Staubli VAL3: TRAJ.pjx

--- TRAJ.pjx ---
Parameters version=s7.5 stackSize=5000 millimeterUnit=true
Program file=changePCircle.pgx
Program file=checkPCircle.pgx
Program file=computeFrame.pgx
Program file=delete.pgx
Program file=deleteItem.pgx
Program file=duplicate.pgx
Program file=find.pgx
Program file=findMove.pgx
Program file=get.pgx
Program file=getDistance.pgx
Program file=getFrame.pgx
Program file=getFrameId.pgx
Program file=getFunctionEdit.pgx
Program file=getFunctionSel.pgx
Program file=getFunctionView.pgx
Program file=getListItem.pgx
Program file=getPoint.pgx
Program file=getSize.pgx
Program file=getSizeItem.pgx
Program file=getTime.pgx
Program file=getTool.pgx
Program file=getTrajItem.pgx
Program file=getTrajType.pgx
Program file=getType.pgx
Program file=goTo.pgx
Program file=HerePoint.pgx
Program file=HerePointCircle.pgx
Program file=insertItem.pgx
Program file=isReachable.pgx
Program file=load.pgx
Program file=loadCycle.pgx
Program file=loadPage.pgx
Program file=makeTraj.pgx
Program file=new.pgx
Program file=onEdit.pgx
Program file=onEditItem.pgx
Program file=onEditTrsf.pgx
Program file=onFunctionEdit.pgx
Program file=onFunctionSel.pgx
Program file=onFunctionView.pgx
Program file=onInsert.pgx
Program file=onProgEnd.pgx
Program file=onRun.pgx
Program file=onSave.pgx
Program file=onStart.pgx
Program file=onStop.pgx
Program file=setFrameId.pgx
Program file=setTool.pgx
Program file=setTrajItem.pgx
Data file=TRAJ.dtx
Library alias=saveData path=Disk://saveData/saveData.pjx
Library alias=page path=Disk://kernel/template/page/page.pjx
Library alias=use path=Disk://kernel/userPage/userPage.pjx
Library alias=language path=Disk://kernel/language/language.pjx
Library alias=tcp path=Disk://kernel/tool/tool.pjx
Library alias=cycleStatus path=Disk://cycleStatus/cycleStatus.pjx
Library alias=pt path=Disk://kernel/template/session/saveTraj/TRAJ/TRAJ.pjx
Type name=TrajectoryItem path=Disk://kernel/template/TrajectoryItem/TrajectoryItem.pjx
Type name=ActionItem path=Disk://kernel/template/ActionItem/ActionItem.pjx
Type name=Trajectory path=Disk://kernel/template/Trajectory/Trajectory.pjx
Type name=InstrItem path=Disk://kernel/template/InstrItem/InstrItem.pjx
Type name=Traies path=Disk://kernel/template/Traies/Traies.pjx
Type name=FrameItem path=Disk://kernel/template/FrameItem/FrameItem.pjx

--- TRAJ.dtx ---
Trajectory tTraj
  [0]
    TrajectoryItem tSuper[3]
      [0]
        num distance
        num moveType = 1
        num nTime
        num nStop
        num nTcpAction
        string comment = "appro"
        bool toStop
        mdesc nom_speed = {tmax=300, rmax=9999, leave=30, reach=30}
        InstrItem iInstr[3]
          [0]
            string sType
            string sData
          [1]
            string sType
            string sData
          [2]
            string sType
            string sData
        num nMoveId
      [1]
        num distance = 2
        num moveType = 1
        num nTime
        num nStop
        num nTcpAction = 2
        string comment = "point"
        bool toStop = true
        mdesc nom_speed = {tmax=300, rmax=9999, leave=30, reach=30}
        InstrItem iInstr[3]
          [0]
            string sType
            string sData
          [1]
            string sType
            string sData
          [2]
            string sType
            string sData
        num nMoveId
      [2]
        num distance
        num moveType = 1
        num nTime
        num nStop
        num nTcpAction
        string comment = "depart"
        bool toStop
        mdesc nom_speed = {tmax=300, rmax=9999, leave=30, reach=30}
        InstrItem iInstr[3]
          [0]
            string sType
            string sData
          [1]
            string sType
            string sData
          [2]
            string sType
            string sData
        num nMoveId
    string sID = "POINT pose"
    num nId
public bool bMoveType[3]
  [0] = true
  [1] = true
  [2] = true
public bool bStepping
bool bToSave
frame fSetFrame = {fatherId=world[0]}
mdesc mMdesc = {accel=10, vel=10, decel=10, blend=off}
string sInstruction
public string sItems
string sMenu[8]
  [5] = "Duplicate"
  [7] = "New"
string sTrajType = "POINT"
pointRx pToGo[2]
  [0] = {fatherId=world[0]}
  [1] = {fatherId=world[0]}
num nFile
pointRx pPoints[3]
  [0] = {fatherId=world[0]}
  [1] = {fatherId=world[0]}
  [2] = {fatherId=world[0]}
Traies pEditPoint
  [0]
    frame fFrame
    num nIndexTool
    string sID
    num nIndexFrame
    TrajItem tData
      [0]
        TrajectoryItem tSuper
          [0]
            num distance
            num moveType
            num nTime
            num nStop
            num nTcpAction
            string comment
            bool toStop
            mdesc nom_speed = {tmax=300, rmax=9999, leave=30, reach=30}
            InstrItem iInstr[3]
              [0]
                string sType
                string sData
              [1]
                string sType
                string sData
              [2]
                string sType
                string sData
            num nMoveId
        pointRx pPoint
        num nType
        pointRx pCircle
string sTrajCycle

--- changePCircle.pgx ---
public program changePCircle(num x_nIndex)
  local bool l_bOk
  local bool l_bRefresh
  local bool l_bUnreach
  local frame l_fTraj
  local joint l_jJoint
  local num l_nIndex
  local num l_nKey
  local num l_nMoveId
  local num l_nResult[2]
  local num l_nView
  local point l_pPoint[2]
  local string l_sButton[2]
  local string l_sEvent
  local string l_sItem
  local string l_sMessage
  local tool l_tTool
  local trsf l_tTrsf
  local trsf l_tTrsfTemp[2]
  local trsf l_trsfPoint
begin
  // INIT
  l_bRefresh=false
  l_nIndex=0
  l_nView=0
  call use:setSizeList(10,3,20,6)
  call use:setView(false)
  // get the tool
  call tcp:getTool(l_tTool,pEditPoint.nIndexTool)
  // get the point and the circle point
  call getPoint(l_pPoint,false,x_nIndex)
  // point final
  pPoints=l_pPoint
  // point intermediare
  pPoints[1]=l_pPoint[1]
  l_tTrsf=l_pPoint[1].trsf
  //
  do
    // check if the intermediate point is reachable
    call isReachable(l_pPoint[1],l_tTool,l_bUnreach)
    //move to
    if cycleStatus:nWorkingMode==1 and !cycleStatus:bCycle and !cycleStatus:bSimulation and !l_bUnreach
      // empty the stack
      resetMotion()
      if distance(here(l_tTool,pEditPoint.fFrame),pPoints[1])>1
        call checkPCircle(x_nIndex,here(l_tTool,pEditPoint.fFrame),l_nResult)
        // CIRCULAR MOVE
        if l_nResult!=-1
          // find P.I. percentage
          call checkPCircle(x_nIndex,pPoints[1],l_nResult[1])
          // take the previous point
          call getPoint(l_pPoint,false,x_nIndex-1)
          //
          // find the intermediate point
          //
          l_pPoint[1]=pPoints[1]
          pPoints[1].trsf=interpolateC(l_pPoint.trsf,pPoints[1].trsf,pPoints.trsf,(l_nResult+l_nResult[1])/2)
          // go to the intermediate point
          pPoints[0]=l_pPoint[1]
          movec(pPoints[1],pPoints,l_tTool,mMdesc)
        else
          // joint MOVE
          movej(pPoints[1],l_tTool,mMdesc)
        endIf
        // joint MOVE
      else
        // joint MOVE
        movej(pPoints[1],l_tTool,mMdesc)
      endIf
    endIf
    // show the menu
    call use:clear(0,13)
    call use:typeMenu(8,"OK")
    if !cycleStatus:bCycle and !cycleStatus:bSimulation
      call use:typeMenu(1,"Here")
    endIf
    // show the context
    call use:listcreate("")
    l_sMessage="coord  X > "+toString(".2",l_tTrsf.x)
    call use:listadd(l_sMessage)
    l_sMessage="coord  Y > "+toString(".2",l_tTrsf.y)
    call use:listadd(l_sMessage)
    l_sMessage="coord  Z > "+toString(".2",l_tTrsf.z)
    call use:listadd(l_sMessage)
    l_sMessage="coord RX > "+toString(".2",l_tTrsf.rx)
    call use:listadd(l_sMessage)
    l_sMessage="coord RY > "+toString(".2",l_tTrsf.ry)
    call use:listadd(l_sMessage)
    l_sMessage="coord RZ > "+toString(".2",l_tTrsf.rz)
    call use:listadd(l_sMessage)
    use:nView=l_nIndex
    call use:listupdate(l_nIndex-l_nView)
    // edit the items
    do
      l_nView=use:nView
      l_nKey=get()
      call use:listevent(l_nKey,l_nIndex,l_sEvent)
      switch l_nKey
        case 271
          // here POINT
          if !cycleStatus:bCycle and !cycleStatus:bSimulation
            // ASK IF YOU WANT TO RECORD THE POINT
            call language:message(l_sMessage,131)
            call language:getYesNo(l_sButton)
            call use:yes_no(l_sMessage,l_sButton,l_bOk)
            if l_bOk
              call HerePointCircle(x_nIndex)
            endIf
          endIf
        break
        case 270
          // clean the line
          call use:listcursor(use:nView,false)
          // EDIT FIELD
          switch l_nIndex
            case 0
              //  x-value
              l_sItem=""
              call use:changeValue(l_tTrsf.x,0,0,2+40-use:nBottomX,use:nView+1+3,l_sItem)
            break
            case 1
              //  y-value
              l_sItem=""
              call use:changeValue(l_tTrsf.y,0,0,2+40-use:nBottomX,use:nView+1+3,l_sItem)
            break
            case 2
              //  z-value
              l_sItem=""
              call use:changeValue(l_tTrsf.z,0,0,2+40-use:nBottomX,use:nView+1+3,l_sItem)
            break
            case 3
              //  rx-value
              l_sItem=""
              call use:changeValue(l_tTrsf.rx,0,0,2+40-use:nBottomX,use:nView+1+3,l_sItem)
            break
            case 4
              //  ry-value
              l_sItem=""
              call use:changeValue(l_tTrsf.ry,0,0,2+40-use:nBottomX,use:nView+1+3,l_sItem)
            break
            case 5
              //  rz-value
              l_sItem=""
              call use:changeValue(l_tTrsf.rz,0,0,2+40-use:nBottomX,use:nView+1+3,l_sItem)
            break
          endSwitch
          l_bRefresh=true
        break
      endSwitch
      delay(0)
    until l_bRefresh==true or l_nKey==255 or l_nKey==278 or l_nKey==271
    //
    // check if is OK   VALUE CHANGE
    //
    if l_nKey==270
      pPoints[1].trsf=l_pPoint[1].trsf=l_tTrsf
    endIf
    //
    l_bRefresh=false
    delay(0)
  until l_nKey==255 or l_nKey==278 or l_nKey==271 or l_bUnreach
  //
  // save the data
  //
  if l_nKey==278
    // record it
    if !l_bUnreach
      // update the circle point
      pEditPoint.tData[x_nIndex].pCircle.trsf=l_tTrsf
    endIf
  endIf
  // release the resource
  call use:nullKey(l_nKey)
end

--- checkPCircle.pgx ---
public program checkPCircle(num x_nIndex, point x_pToCheck, num& x_nResult[])
  local num i
  local bool l_bDistance[3]
  local bool l_bUnreach
  local frame l_fFrame
  local num l_nDistance
  local num l_nNewDist
  local num l_nStep
  local num l_nTo
  local point l_pCircle[3]
  local point l_pPoint
  local tool l_tTool
begin
  // check if the x_pToCheck is inside the Circle
  //
  //  INIT
  //
  l_nDistance=1000
  l_nStep=x_nResult=-1
  call tcp:getTool(l_tTool,pEditPoint.nIndexTool)
  l_pPoint=here(l_tTool,pEditPoint.fFrame)
  // get the three point
  if x_nIndex>0
    call getPoint(l_pCircle,false,x_nIndex-1)
    call getPoint(l_pCircle[1],false,x_nIndex)
  endIf
  // check if the points are the same
  l_bDistance=distance(position(l_pCircle,pEditPoint.fFrame),position(l_pCircle[2],pEditPoint.fFrame))<1
  l_bDistance[1]=distance(position(l_pCircle[1],pEditPoint.fFrame),position(l_pCircle[2],pEditPoint.fFrame))<1
  l_bDistance[2]=distance(position(l_pCircle,pEditPoint.fFrame),position(l_pCircle[1],pEditPoint.fFrame))<1
  call isReachable(l_pCircle,l_tTool,l_bUnreach)
  if !l_bUnreach
    call isReachable(l_pCircle[1],l_tTool,l_bUnreach)
    // check the frame
    if !l_bUnreach
      l_bUnreach=setFrame(l_pCircle,l_pCircle[2],l_pCircle[1],fSetFrame)!=0
    endIf
  endIf
  if l_bDistance or l_bDistance[1] or l_bDistance[2] or l_bUnreach
    // not valid circle point
    x_nResult=-1
    return
  endIf
  // first check step 0.1
  for i=0 to 1 step 0.1
    l_pPoint.trsf=interpolateC(position(l_pCircle,pEditPoint.fFrame),position(l_pCircle[2],pEditPoint.fFrame),position(l_pCircle[1],pEditPoint.fFrame),i)
    l_nNewDist=distance(x_pToCheck.trsf,l_pPoint.trsf)
    if l_nNewDist<l_nDistance
      l_nDistance=l_nNewDist
      l_nStep=i
    endIf
  endFor
  if l_nStep!=-1
    // second step 0.01
    l_nTo=min(l_nStep+0.05,1)
    for i=max(l_nStep-0.05,0) to l_nTo step 0.01
      l_pPoint.trsf=interpolateC(position(l_pCircle,pEditPoint.fFrame),position(l_pCircle[2],pEditPoint.fFrame),position(l_pCircle[1],pEditPoint.fFrame),i)
      l_nNewDist=distance(x_pToCheck.trsf,l_pPoint.trsf)
      if l_nNewDist<l_nDistance
        l_nDistance=l_nNewDist
        l_nStep=i
      endIf
    endFor
  endIf
  if l_nStep!=-1
    // third step 0.001
    l_nTo=min(l_nStep+0.005,1)
    for i=max(l_nStep-0.005,0) to l_nTo step 0.001
      l_pPoint.trsf=interpolateC(position(l_pCircle,pEditPoint.fFrame),position(l_pCircle[2],pEditPoint.fFrame),position(l_pCircle[1],pEditPoint.fFrame),i)
      l_nNewDist=distance(x_pToCheck.trsf,l_pPoint.trsf)
      if l_nNewDist<l_nDistance
        l_nDistance=l_nNewDist
        l_nStep=i
      endIf
    endFor
  endIf
  // 5 mm tollerance
  if l_nDistance<=5
    // store the value
    x_nResult=l_nStep
  endIf
end

--- computeFrame.pgx ---
public program computeFrame(num x_nNewFrame)
  local num i
begin
    // recompute all the point into the new frame
  for i=0 to size(pEditPoint.tData)-1
    pEditPoint.tData[i].pPoint.trsf=position(pEditPoint.tData[i].pPoint,saveData:fFrameItem[x_nNewFrame].fFrame)
  endFor
end

--- delete.pgx ---
public program delete(string x_sName, num& x_nResult[])
  local string l_sItem
  local num l_nSize
begin
  //
  // delete the select trajectory
  //
  if isDefined(pt:tTraj[x_sName])
    // delete
    delete(pt:tTraj[x_sName])
    // save it
    bToSave=true
    x_nResult=0
  else
    x_nResult=-1
  endIf
end

--- deleteItem.pgx ---
public program deleteItem(num& x_nIndex)
  local num i
  local string l_sItem
begin
  // delete the selected item
    // delete all the field
    delete(pEditPoint.tData[x_nIndex])
end

--- find.pgx ---
public program find(string& x_sItem[], bool& x_bFound[])
begin
  // check if the item has been found
  x_bFound=isDefined(pt:tTraj[x_sItem])
end

--- findMove.pgx ---
public program findMove(num x_nIndex, tool x_tTool, num& x_nMoveType[])
  local point l_pHere
  local num l_nResult
  local num l_nIndexTool
  local num l_nSize
  local num l_nMoveType
  local point l_pPoint[2]
  local joint l_jHere
  local bool l_bUnreach
begin
  //
  // MOVE TO THE POINT
  //
  // get all the value that you need
  call getSizeItem(false,l_nSize)
  l_pHere=here(x_tTool,pEditPoint.fFrame)
  // get the point and the circle point
  call getPoint(pPoints,false,x_nIndex)
  call getPoint(l_pPoint,false,x_nIndex)
  pPoints[1].trsf=position(l_pPoint,pEditPoint.fFrame)
  pPoints[2].trsf={0,0,0,0,0,0}
  // take the moveType for the x_nIndex
  l_nMoveType=x_nMoveType
  // Set to JOINT for default
  x_nMoveType=0
  //
  // LOOK FOR CIRCLE MOVE
  //
  if distance(l_pHere,pPoints[1])>1
    if x_nIndex>0 and l_nMoveType==2
      // FORWARD
      call getPoint(l_pPoint,false,x_nIndex-1)
      pPoints.trsf=position(l_pPoint,pEditPoint.fFrame)
      if distance(l_pHere,pPoints)<1
        // move circular forward
        x_nMoveType=2
      else
        // look if is it inside the traiectory
        call checkPCircle(x_nIndex,here(x_tTool,pEditPoint.fFrame),l_nResult)
        if l_nResult!=-1 and l_nResult!=0 and l_nResult!=1
          // save the percentage inside the type
          x_nMoveType=2+l_nResult
        endIf
      endIf
    endIf
    if x_nIndex<(l_nSize-1) and x_nMoveType==0
      // BACKWARD
      l_nMoveType=pEditPoint.tData[x_nIndex+1].tSuper.moveType
      if l_nMoveType==2
        // get the point and the circle point
        call getPoint(l_pPoint,false,x_nIndex+1)
        pPoints.trsf=position(l_pPoint,pEditPoint.fFrame)
        if distance(l_pHere,pPoints)<1
          // move circular backward
          x_nMoveType=-2
        else
          // look if is it inside the traiectory
          call checkPCircle(x_nIndex+1,here(x_tTool,pEditPoint.fFrame),l_nResult)
          if l_nResult!=-1 and l_nResult!=0 and l_nResult!=1
            // save the percentage inside the type
            x_nMoveType=-2-l_nResult
          endIf
        endIf
      endIf
    endIf
  endIf
  //
  // NO CIRCLE
  //
  if abs(x_nMoveType)<2
    l_nMoveType=pEditPoint.tData[x_nIndex].tSuper.moveType
    //
    // move forward
    //
    if x_nIndex>0 and l_nMoveType==1
      // get the point and the circle point
      call getPoint(l_pPoint,false,x_nIndex-1)
      pPoints.trsf=position(l_pPoint,pEditPoint.fFrame)
      if distance(l_pHere,pPoints)<1
        // set to linear
        x_nMoveType=1
      elseIf setFrame(pPoints,pPoints[1],pPoints[2],fSetFrame)==0
        // check frame
        l_pHere=here(x_tTool,fSetFrame)
        pPoints[1].trsf=position(pPoints[1],fSetFrame)
        if l_pHere.trsf.x>=0 and l_pHere.trsf.x<=pPoints[1].trsf.x and abs(l_pHere.trsf.y)<1 and abs(l_pHere.trsf.z)<1
          // set to linear
          x_nMoveType=1
        endIf
      endIf
    endIf
    //
    // move back
    //
    if x_nIndex<(l_nSize-1) and x_nMoveType!=1
      l_nMoveType=pEditPoint.tData[x_nIndex+1].tSuper.moveType
      if l_nMoveType==1
        // get the point and the circle point
        call getPoint(l_pPoint,false,x_nIndex)
        pPoints[1].trsf=position(l_pPoint,pEditPoint.fFrame)
        // get the point and the circle point
        call getPoint(l_pPoint,false,x_nIndex+1)
        pPoints.trsf=position(l_pPoint,pEditPoint.fFrame)
        if distance(l_pHere,pPoints)<1
          // switch to linear
          x_nMoveType=1
        elseIf setFrame(pPoints,pPoints[1],pPoints[2],fSetFrame)==0
          // check frame
          l_pHere=here(x_tTool,fSetFrame)
          pPoints[1].trsf=position(pPoints[1],fSetFrame)
          if l_pHere.trsf.x>=0 and l_pHere.trsf.x<=pPoints[1].trsf.x and abs(l_pHere.trsf.y)<1 and abs(l_pHere.trsf.z)<1
            // set to linear
            x_nMoveType=1
          endIf
        endIf
      endIf
    endIf
  endIf
end

--- getDistance.pgx ---
public program getDistance(tool x_tTool (dimensions=1), num& x_nDistance[] (dimensions=1), bool x_bCycle (dimensions=1), num x_nIndex (dimensions=1))
  local num l_nValue
  local point l_pActual
  local point l_pPoint
  local point l_pPrev
  local trsf l_trsfEmpty
begin
  // first point
  if x_nIndex==0
    x_nDistance=10
    return
  else
    //
    // get the point
    //
    call getPoint(l_pActual,x_bCycle,x_nIndex)
    call getPoint(l_pPrev,x_bCycle,x_nIndex-1)
    if x_bCycle
      x_nDistance=distance(l_pPrev.trsf,l_trsfEmpty)
    else
      x_nDistance=distance(l_pPrev.trsf,l_trsfEmpty)
    endIf
  endIf
end

--- getFunctionEdit.pgx ---
public program getFunctionEdit(string& x_sName[])
  local string l_sMessage
begin
  //
  // define your message for the
  // function KEY
  //
  // NOTE is an ARRAY[0..7]
  //
  // example:
  // x_sName[1]="DEMO"
  // active the F2 button
  //
  // HERE
  call language:message(l_sMessage,150)
  x_sName[0]=l_sMessage
  // ALIGN
  call language:message(l_sMessage,134)
  x_sName[1]=l_sMessage
end

--- getFunctionSel.pgx ---
public program getFunctionSel(string& x_sName[])
  local string l_sMessage
begin
  //
  // define your message for the
  // function KEY
  //
  // NOTE is an ARRAY[0..7]
  //
  // example:
  // x_sName[1]="DEMO"
  // active the F2 button
  //
end

--- getFunctionView.pgx ---
public program getFunctionView(string& x_sName[])
  local string l_sMessage
begin
  //
  // define your message for the
  // function KEY
  //
  // NOTE is an ARRAY[0..7]
  //
  // example:
  // x_sName[1]="DEMO"
  // active the F2 button
  //
  // HERE
  call language:message(l_sMessage,150)
  x_sName[0]=l_sMessage
  // ALIGN
  call language:message(l_sMessage,134)
  x_sName[1]=l_sMessage
end

--- getListItem.pgx ---
public program getListItem(string& x_sItem[], num x_nIndex)
  local trsf l_tTrsf
  local string l_sItem[6]
  local string l_sEvent
  local string l_sItem2[7]
begin
  //
  // define the item to show in the edit page Traj
  // customize an array and copy to x_sItem...
  //
  // see other traj as example
  // take it
  l_sEvent="coord  "
  l_tTrsf=pEditPoint.tData[x_nIndex].pPoint.trsf
  // show them
  l_sItem[0]=l_sItem2[0]=("coord  X > "+toString(".2",l_tTrsf.x))
  l_sItem[1]=l_sItem2[1]=("coord  Y > "+toString(".2",l_tTrsf.y))
  l_sItem[2]=l_sItem2[2]=("coord  Z > "+toString(".2",l_tTrsf.z))
  l_sItem[3]=l_sItem2[3]=("coord RX > "+toString(".2",l_tTrsf.rx))
  l_sItem[4]=l_sItem2[4]=("coord RY > "+toString(".2",l_tTrsf.ry))
  l_sItem[5]=l_sItem2[5]=("coord RZ > "+toString(".2",l_tTrsf.rz))
  // check the moveType
  if pEditPoint.tData[x_nIndex].tSuper.moveType==2
    // insert the circle POINT
    l_sItem2[6]="Point intermediate"
    call use:stringCopy(l_sItem2,x_sItem)
  else
    // look for intermediate point
    call use:stringCopy(l_sItem,x_sItem)
  endIf
end

--- getPoint.pgx ---
public program getPoint(point& x_pPoint[], bool x_bCycle, num x_nIndex)
  local string l_sItem
  local num l_nSize
  local num i
  local num l_nPoint
begin
  // take
  if x_bCycle
    // real point
    x_pPoint=pt:tTraj[sTrajCycle].tData[x_nIndex].pPoint
    if size(x_pPoint)>1
      x_pPoint[1]=pt:tTraj[sTrajCycle].tData[x_nIndex].pCircle
    endIf
  else
    // edit point
    x_pPoint=pEditPoint.tData[x_nIndex].pPoint
    if size(x_pPoint)>1
      x_pPoint[1]=pEditPoint.tData[x_nIndex].pCircle
    endIf
  endIf
end

--- getSizeItem.pgx ---
public program getSizeItem(bool x_bCycle, num& x_nSize)
  local string l_sType
  local string l_sKey
  local num i
begin
  //
  // get the size of the collection
  //
  if x_bCycle
    x_nSize=size(pt:tTraj[sTrajCycle].tData)
  else
    x_nSize=size(pEditPoint.tData)
  endIf
end

--- getTime.pgx ---
public program getTime(num& x_nTime[], bool x_bCycle, num x_nIndex)
begin
  // get the time DATA
  if x_bCycle
    // get the time DATA
    x_nTime=pt:tTraj[sTrajCycle].tData[x_nIndex].tSuper.nTime
  else
    // get the time DATA
    x_nTime=pEditPoint.tData[x_nIndex].tSuper.nTime
  endIf
end

--- getTrajType.pgx ---
program getTrajType(string& x_sTrajType[])
  local num l_nPos
  local string l_sPath
begin
  // get the trajType
  l_sPath=libPath()
  if find(l_sPath,sTrajType)==-1 or sTrajType==""
    do
      l_nPos=find(l_sPath,"/")
      if l_nPos==-1
        l_nPos=find(l_sPath,"\")
      endIf
      if l_nPos!=-1
        l_sPath=right(l_sPath,len(l_sPath)-l_nPos-1)
      endIf
    until l_nPos==-1
    //
    sTrajType=l_sPath
  endIf
  // return back
  x_sTrajType=sTrajType
end

--- goTo.pgx ---
public program goTo(tool x_tTool, mdesc x_mDesc, num x_nMoveType, bool& x_bUnreached[], num x_nIndex)
  local point l_pTrsf
  local bool l_bInside
  local tool l_tTool
  local point l_pHere
  local string l_sMessage
  local num l_nSize
  local num i
  local mdesc l_mSpeed
  local joint l_jJoint
  local point l_pPoint[2]
  local bool l_bUnreach
begin
  // get the moveType
  call findMove(x_nIndex,x_tTool,x_nMoveType)
  if isEmpty()
    // get the POINT
    call getPoint(l_pPoint,false,x_nIndex)
    pToGo=l_pPoint
    pToGo[1]=l_pPoint[1]
    l_pHere=here(x_tTool,pEditPoint.fFrame)
    // step by step motion
    if x_nMoveType==0
      // or is not in range
      movej(pToGo,x_tTool,x_mDesc)
    elseIf x_nMoveType==1
      movel(pToGo,x_tTool,x_mDesc)
    elseIf x_nMoveType>2
      // inside the trajectory
      // take the percentage arcInterpo
      call getPoint(l_pPoint,false,x_nIndex-1)
      call isReachable(pToGo,x_tTool,l_bUnreach)
      if !l_bUnreach and pointToJoint(x_tTool,herej(),l_pPoint,l_jJoint)
        pToGo[1].trsf=interpolateC(position(l_pPoint,pEditPoint.fFrame),pToGo[1].trsf,pToGo.trsf,(1-(2-x_nMoveType))/2)
      endIf
    elseIf x_nMoveType<=-2
      // move circular backward
      call getPoint(l_pPoint,false,x_nIndex+1)
      call isReachable(l_pPoint,x_tTool,l_bUnreach)
      if !l_bUnreach
        // look for percentage value need
        if x_nMoveType==-2
          pToGo[1].trsf=position(l_pPoint[1],pEditPoint.fFrame)
        else
          pToGo[1].trsf=interpolateC(pToGo.trsf,position(l_pPoint[1],pEditPoint.fFrame),position(l_pPoint,pEditPoint.fFrame),(abs(x_nMoveType+2))/2)
        endIf
      endIf
    endIf
    if l_bUnreach
      // get the message point is not reachable
      call language:message(l_sMessage,-5)
      call use:type(0,12,"!!! "+l_sMessage)
    elseIf x_nMoveType!=0 and x_nMoveType!=1
      // CIRCULAR MOVE
      movec(pToGo[1],pToGo,x_tTool,x_mDesc)
    endIf
  endIf
end

--- HerePoint.pgx ---
public program HerePoint(num x_nIndex)
  local tool l_tTool
  local point l_pHere
  local frame l_fFrame
  local num i
  local num l_nIndex
  local num l_nSize
begin
  //
  // take the point
  //
  // frame
  call getFrame(fSetFrame,false)
  // tool
  call tcp:getTool(l_tTool,pEditPoint.nIndexTool)
  // here
  l_pHere=here(l_tTool,fSetFrame)
  resetMotion()
  // save the trsf
  pEditPoint.tData[x_nIndex].pPoint.trsf=l_pHere.trsf
  // check the moveType to save the config
  if pEditPoint.tData[x_nIndex].tSuper.moveType==0
    pEditPoint.tData[x_nIndex].pPoint.config=l_pHere.config
  endIf
  // to be save

end

--- HerePointCircle.pgx ---
public program HerePointCircle(num x_nIndex)
  local tool l_tTool
  local point l_pHere
  local frame l_fFrame
  local num i
  local num l_nIndex
  local num l_nSize
begin
  //
  // take the point
  //
  // frame
  call getFrame(fSetFrame,false)
  // tool
  call tcp:getTool(l_tTool,pEditPoint.nIndexTool)
  // here
  l_pHere=here(l_tTool,fSetFrame)
  resetMotion()
  // save the trsf
  pEditPoint.tData[x_nIndex].pCircle.trsf=l_pHere.trsf
  // check the moveType to save the config
  if pEditPoint.tData[x_nIndex].tSuper.moveType==0
    pEditPoint.tData[x_nIndex].pCircle.config=l_pHere.config
  endIf
end

--- insertItem.pgx ---
public program insertItem(num& x_nIndexCopy, num x_nIndexPaste)
  local num l_nLastType
  local point l_pPoint
  local num l_nType
begin
  //
  // use to add more elements from the typical one
  //
  // insert all the field
  //
  l_pPoint=pEditPoint.tData[x_nIndexCopy].pPoint
  l_nLastType=pEditPoint.tData[x_nIndexCopy].nType
  if l_nLastType==0
    l_nType=0
  elseIf l_nLastType==2 or l_nLastType==1
    l_nType=2
  endIf
  insert(pEditPoint.tData[x_nIndexPaste])
  // set IT - link it
  link(pEditPoint.tData[x_nIndexPaste].pPoint,pEditPoint.fFrame)
  link(pEditPoint.tData[x_nIndexPaste].pCircle,pEditPoint.fFrame)
  pEditPoint.tData[x_nIndexPaste].pPoint.trsf=l_pPoint.trsf
  // set IT
  pEditPoint.tData[x_nIndexPaste].nType=l_nType
end

--- isReachable.pgx ---
program isReachable(pointRx& x_pPoint[], tool x_tTool, bool& x_bUnreached)
  local joint l_jJoint
  local point l_pPoint
begin
  // check the point...
  if pointToJoint(x_tTool,herej(),x_pPoint,l_jJoint)
    x_bUnreached=false
    if size(x_pPoint)>1 and pointToJoint(x_tTool,herej(),x_pPoint[1],l_jJoint)
      x_bUnreached=false
    elseIf size(x_pPoint)>1
      x_bUnreached=true
    endIf
  else
    x_bUnreached=true
  endIf

end

--- load.pgx ---
public program load(string x_sItem (dimensions=1), num& x_nResult (dimensions=1))
  local num i
  local string l_sMessage
  local string l_sType
begin
  // load the select trajectory..already loaded
  call getTrajType(l_sType)
  if find(pt:libPath(),saveData:sPathTraj)==-1
    pt:libLoad(saveData:sPathTraj+l_sType)
    delay(0)
    if saveData:bDebug
      ? "loading TRAJ..."+saveData:sPathTraj+l_sType
    endIf
  endIf
  // use the type...
  if isDefined(pt:tTraj[x_sItem])
    // link the frame and all the points
    call pt:link_all(x_sItem)
    // check if link and defined
    pEditPoint=pt:tTraj[x_sItem]
    // link all
    link(pEditPoint.fFrame,world)
    for i=0 to size(pEditPoint.tData)-1
      link(pEditPoint.tData[i].pPoint,pEditPoint.fFrame)
      link(pEditPoint.tData[i].pCircle,pEditPoint.fFrame)
    endFor
    pEditPoint.sID=x_sItem
  elseIf x_sItem!=""
    // not FOUND
    call language:message(l_sMessage,-7)
    x_nResult=-1
    popUpMsg(l_sMessage+x_sItem)
  endIf
end

--- loadCycle.pgx ---
public program loadCycle(string x_sItem, num& x_nResult[])
  local string l_sType
  local string l_sMessage
begin
  // load the select trajectory..already loaded
  call getTrajType(l_sType)
  if find(pt:libPath(),saveData:sPathTraj)==-1
    pt:libLoad(saveData:sPathTraj+l_sType)
    delay(0)
    if saveData:bDebug
      ? "loading TRAJ..."+saveData:sPathTraj+l_sType
    endIf
  endIf
  // use the type...
  if isDefined(pt:tTraj[x_sItem])
    // link the frame and all the points
    call pt:link_all(x_sItem)
    sTrajCycle=x_sItem

  else
    // not FOUND
    call language:message(l_sMessage,-7)
    x_nResult=-1
    cycleStatus:bToStop=true
    popUpMsg(l_sMessage+x_sItem)
  endIf
end

--- makeTraj.pgx ---
public program makeTraj(string& x_sItem[])
  local num i
  local num l_nDistance
  local num l_nSize
  local tool l_tTool
  local bool l_bToStop
  local mdesc l_mDesc
  local num l_nMoveId
  local bool l_bOk
  local string l_sType
  local TrajectoryItem l_tTraj
  local ActionItem l_aAction
  local point l_pPoint[2]
begin
  // take the TOOL
  call tcp:getTool(l_tTool,pt:tTraj[sTrajCycle].nIndexTool)
  // the maximum size
  call getSizeItem(true,l_nSize)
  //
  // for all of my traj cyclePoints move the robot
  //
  resize(tTraj.tSuper,1,size(pt:tTraj[sTrajCycle].tData))
  for i=0 to (l_nSize-1)
    tTraj.tSuper[i]=pt:tTraj[sTrajCycle].tData[i].tSuper
  endFor
  tTraj.sID="TRAJ "+pt:tTraj[sTrajCycle].sID
  call cycleStatus:addTraj(tTraj)
  //
  // for all of my traj cyclePoints move the robot
  //
  for i=0 to (l_nSize-1)
    //
    // get the point info
    //
    l_tTraj=pt:tTraj[sTrajCycle].tData[i].tSuper
    call getPoint(l_pPoint,true,i)
    //
    // get the distance in percentage
    call getDistance(l_tTool,l_nDistance,true,i)
    //
    // give to the traj library the percentage distance
    //
    if l_bToStop
      l_tTraj.nom_speed.blend=off
    elseIf l_tTraj.moveType!=0
      l_tTraj.nom_speed.blend=Cartesian
    endIf
    //
    // put the move in the stack
    //
    switch l_tTraj.moveType
      case 0
        // or is not in range
        l_nMoveId=movej(l_pPoint,l_tTool,l_tTraj.nom_speed)
      break
      case 1
        l_nMoveId=movel(l_pPoint,l_tTool,l_tTraj.nom_speed)
      break
      case 2
        l_nMoveId=movec(l_pPoint[1],l_pPoint,l_tTool,l_tTraj.nom_speed)
      break
    endSwitch
    //
    // set the ID
    //
    l_aAction.nDistance=l_nDistance
    l_aAction.nPointId=i
    l_aAction.nMoveId=l_nMoveId
    l_aAction.sIdTraj="TRAJ "+pt:tTraj[sTrajCycle].sID
    call cycleStatus:putInstr_Traj(l_aAction,l_tTraj,pt:tTraj[sTrajCycle].nIndexTool,l_nSize)
    // there is a waitEndMove
    if l_tTraj.toStop
      waitEndMove()
      delay(l_tTraj.nStop)
      // wait all the action has been done
      wait(cycleStatus:bActionRunning==false)
    endIf
  endFor
  // bye bye
end

--- onEditItem.pgx ---
public program onEditItem(string& x_sEvent[], num x_nIndex, num x_nIndexItem)
begin
  if x_nIndex!=6
    // edit the custom element that was add in the list
    call onEditTrsf(x_nIndex,x_nIndexItem,x_sEvent)
  elseIf x_nIndex==6
    call changePCircle(x_nIndexItem)
  endIf
end

--- onEditTrsf.pgx ---
public program onEditTrsf(num x_nIndex, num x_nIndexItem, string x_sEvent)
  local num i
  local num l_nMin
  local num l_nMax
  local trsf l_tTrsf
  local string l_sEmpty
  local num l_nOldValue
  local num l_nNewValue
  local string l_sMessage
begin
  //  if $fileExists("changePoint.txt")
  //    nFile=$fileOpen("changePoint.txt","a")
  //  else
  //    nFile=$fileOpen("changePoint.txt","w")
  //  endIf
  // edit TRSF OF THE POINT
  l_tTrsf=pEditPoint.tData[x_nIndexItem].pPoint.trsf
  // find the >
  call use:findPos(x_sEvent,">",i)
  i=i+1
  // find the line
  if !cycleStatus:bCycle
    l_nMin=l_nMax=0
  else
    switch x_nIndex
      case 0
        // x
        l_nMin=l_tTrsf.x-10
        l_nMax=l_tTrsf.x+10
      break
      case 1
        // y
        l_nMin=l_tTrsf.y-10
        l_nMax=l_tTrsf.y+10
      break
      case 2
        // z
        l_nMin=l_tTrsf.z-10
        l_nMax=l_tTrsf.z+10
      break
      case 3
        // rx
        l_nMin=l_tTrsf.rx-5
        l_nMax=l_tTrsf.rx+5
      break
      case 4
        // ry
        l_nMin=l_tTrsf.ry-5
        l_nMax=l_tTrsf.ry+5
      break
      case 5
        // rz
        l_nMin=l_tTrsf.rz-5
        l_nMax=l_tTrsf.rz+5
      break
    endSwitch
  endIf
  // clean the line
  call use:listcursor(use:nView,false)
  //
  switch x_nIndex
    case 0
      //  x-value
      l_nOldValue=l_tTrsf.x
      call use:changeValue(l_tTrsf.x,l_nMin,l_nMax,i+40-use:nBottomX,use:nView+1,l_sEmpty)
      l_nNewValue=l_tTrsf.x
    break
    case 1
      //  y-value
      l_nOldValue=l_tTrsf.y
      call use:changeValue(l_tTrsf.y,l_nMin,l_nMax,i+40-use:nBottomX,use:nView+1,l_sEmpty)
      l_nNewValue=l_tTrsf.y
    break
    case 2
      //  z-value
      l_nOldValue=l_tTrsf.z
      call use:changeValue(l_tTrsf.z,l_nMin,l_nMax,i+40-use:nBottomX,use:nView+1,l_sEmpty)
      l_nNewValue=l_tTrsf.z
    break
    case 3
      //  rx-value
      l_nOldValue=l_tTrsf.rx
      call use:changeValue(l_tTrsf.rx,l_nMin,l_nMax,i+40-use:nBottomX,use:nView+1,l_sEmpty)
      l_nNewValue=l_tTrsf.rx
    break
    case 4
      //  ry-value
      l_nOldValue=l_tTrsf.ry
      call use:changeValue(l_tTrsf.ry,l_nMin,l_nMax,i+40-use:nBottomX,use:nView+1,l_sEmpty)
      l_nNewValue=l_tTrsf.ry
    break
    case 5
      //  rz-value
      l_nOldValue=l_tTrsf.rz
      call use:changeValue(l_tTrsf.rz,l_nMin,l_nMax,i+40-use:nBottomX,use:nView+1,l_sEmpty)
      l_nNewValue=l_tTrsf.rz
    break
  endSwitch
  // validate
  if !use:bUseEscape
    pEditPoint.tData[x_nIndexItem].pPoint.trsf=l_tTrsf
    //    // save it into a file
    //    if l_nNewValue!=l_nOldValue
    //      l_sMessage=getDate(" %d %m %Y %H:%M:%S")
    //      l_sMessage=l_sMessage+" Change TRAJ: "+ pEditPoint.sID+", index: "+toString(l_sEmpty,x_nIndexItem+1)+" , name: "+ pEditPoint.tData[x_nIndexItem].tSuper.comment+" , "+ x_sEvent+" to: "+toString(".3",l_nNewValue)
    //      $fileSet(nFile,l_sMessage,1)
    //    endIf
  endIf
end

--- onFunctionEdit.pgx ---
public program onFunctionEdit(num x_nIndex, string x_sEvent, num x_nFunctionKey)
  local string l_sMessage
  local string l_sButton[2]
  local bool l_bOk
  local string l_sPage
  local string l_sItem
  local tool l_tTool
  local point l_pAlign
  local bool l_bYes
  local string l_sMessage2
begin
  //
  // do on Key action
  //
  // x_nIndex = actual index item
  // x_sEvent = actual event item
  //
  switch x_nFunctionKey
    // F1 button
    case 271
      // HERE POINT
      if !cycleStatus:bCycle
        if x_sEvent!="Point intermediate"
          call language:message(l_sMessage,160)
          call language:getYesNo(l_sButton)
          call use:yes_no(l_sMessage,l_sButton,l_bYes)
          if l_bYes
            call HerePoint(x_nIndex)
          endIf
        else
          call language:message(l_sMessage,131)
          call language:getYesNo(l_sButton)
          call use:yes_no(l_sMessage,l_sButton,l_bYes)
          if l_bYes
            call HerePointCircle(x_nIndex)
          endIf
        endIf
        bToSave=true
      endIf
    break
    // F2 button
    case 272
      // ALIGN
      if !cycleStatus:bCycle
        resetMotion()
        call getFrame(fSetFrame,false)
        // tool
        call tcp:getTool(l_tTool,pEditPoint.nIndexTool)
        l_pAlign=here(l_tTool,world)
        l_pAlign.trsf=align(l_pAlign.trsf,fSetFrame.trsf)
        call language:message(l_sMessage,203)
        call language:message(l_sMessage2,134)
        l_sMessage=l_sMessage+" "+l_sMessage2+"..."
        call use:timerDialog(l_sMessage,0)
        movel(l_pAlign,l_tTool,mMdesc)
        watch(isEmpty() or isKeyPressed(255),3)
        delay(1)
      endIf
    break
    // F3 button
    case 273
    break
    // F4 button
    case 274
    break
    // F5 button
    case 275
    break
    // F6 button
    case 276
    break
    // F7 button
    case 277
    break
    // F8 button
    case 278
      // save it
      bToSave=true
    break
  endSwitch
end

--- onFunctionSel.pgx ---
public program onFunctionSel(num x_nIndex, string x_sEvent, num x_nFunctionKey)
begin
  //
  // do on Key action
  //
  // x_nIndex = actual index item
  // x_sEvent = actual event item
  //
  switch x_nFunctionKey
    // F1 button
    case 271
    break
    // F2 button
    case 272
    break
    // F3 button
    case 273
    break
    // F4 button
    case 274
    break
    // F5 button
    case 275
    break
    // F6 button
    case 276
    break
    // F7 button
    case 277
    break
    // F8 button
    case 278
    break
  endSwitch
end

--- onFunctionView.pgx ---
public program onFunctionView(num x_nIndex, string x_sEvent, num x_nFunctionKey)
  local string l_sMessage
  local string l_sButton[2]
  local bool l_bYes
  local tool l_tTool
  local point l_pAlign
  local string l_sMessage2
  local joint l_jJoint
begin
  //
  // do on Key action
  //
  // x_nIndex = actual index item
  // x_sEvent = actual event item
  //
  switch x_nFunctionKey
    // F1 button
    case 271
      // HERE POINT
      if !cycleStatus:bCycle
        call language:message(l_sMessage,160)
        call language:getYesNo(l_sButton)
        call use:yes_no(l_sMessage,l_sButton,l_bYes)
        if l_bYes
          call HerePoint(x_nIndex)
        endIf
        bToSave=true
      endIf
    break
    // F2 button
    case 272
      // ALIGN
      if !cycleStatus:bCycle and !cycleStatus:bSimulation
        resetMotion()
        call getFrame(fSetFrame,false)
        // tool
        call tcp:getTool(l_tTool,pEditPoint.nIndexTool)
        l_pAlign=here(l_tTool,world)
        l_pAlign.trsf=align(l_pAlign.trsf,fSetFrame.trsf)
        // check the align
        if pointToJoint(l_tTool,herej(),l_pAlign,l_jJoint)
          call language:message(l_sMessage,203)
          call language:message(l_sMessage2,134)
          l_sMessage=l_sMessage+" "+l_sMessage2+"..."
          call use:timerDialog(l_sMessage,0)
          movej(l_pAlign,l_tTool,mMdesc)
          watch(isEmpty() or isKeyPressed(255),3)
          if !isEmpty()
            resetMotion()
          endIf
          delay(2)
        endIf
      endIf
    break
    // F3 button
    case 273
    break
    // F4 button
    case 274
    break
    // F5 button
    case 275
    break
    // F6 button
    case 276
    break
    // F7 button
    case 277
    break
    // F8 button
    case 278
    break
  endSwitch
end

--- onInsert.pgx ---
public program onInsert(string& x_sItem[])
  local string l_sEvent
  local num l_nKey
  local num l_nIndex
  local num l_nSize
  local num i
  local string l_sMessage
  local bool l_bFound
  local string l_sType
  local bool l_bUseFilter
  local string l_sPaste
  local num l_nResult
  local num l_nX
  local num l_nY
  local string l_sName
begin
  // get the type
  call getTrajType(x_sItem)
  saveData:sTrajTypeUsing=x_sItem
  cls()
  // is a filter using ??
  if saveData:sTrajFilter!=""
    l_bUseFilter=true
    call language:message(l_sMessage,64)
    call use:type(0,1,l_sMessage+">ON")
  else
    // clean
    call use:typeLen(0,1," ",use:nBottomX)
  endIf
  //
  // CREATE THE LIST
  //
  // define your list size for default
  call use:setSizeList(19,0,19,11)
  call use:setView(false)
  call use:listcreate(x_sItem)
  // take the coordinate....
  l_nX=40-use:nBottomX-1
  l_nY=use:nBottomY+1
  // show the message
  call language:message(l_sMessage,61)
  call use:stringToArray(l_sMessage,sMenu)
  call use:setMenu(sMenu,true,3)
  // Build the list
  call getSize(l_nSize)
  for i=0 to l_nSize-1
    call get(l_sEvent,i)
    if l_sEvent!=""
      //
      // use the filter ?
      //
      // check if the bProcessList filter is active
      //
      l_bFound=true
      if saveData:sTrajFilter!=""
        l_bFound=find(l_sEvent,saveData:sTrajFilter)!=-1
      endIf
      // add
      if l_bFound
        call use:listadd(l_sEvent)
      endIf
    endIf
  endFor
  call use:listupdate(0)
  do
    // get the item
    l_nKey=get()
    call use:listevent(l_nKey,l_nIndex,l_sEvent)
    if l_nKey==271 and l_bUseFilter
      // Build the list
      call getSize(l_nSize)
      // empty and rebuild
      call use:listempty()
      for i=0 to l_nSize-1
        call get(l_sEvent,i)
        if l_sEvent!=""
          call use:listadd(l_sEvent)
        endIf
      endFor
      // clean
      call use:typeLen(0,1," ",use:nBottomX)
      call use:typeMenu(1," ")
      l_bUseFilter=false
      call use:listupdate(0)
    endIf
    //
  until l_nKey==270 or l_nKey==255 or l_nKey==278 or l_nKey==276
  //
  switch l_nKey
    case 270
      // save the name
      l_sName=l_sEvent
    break
    case 276
      // duplicate
      // ask for the new
      call language:message(l_sMessage,21)
      call use:type(l_nX,l_nY,l_sMessage)
      l_sName=l_sEvent
      // read the new trajectory
      call use:read(l_nX+len(l_sMessage),l_nY,l_sName,10,false)
      if !use:bUseEscape
        call duplicate(l_sEvent,l_sName,l_nResult)
      endIf
    break
    case 278
      call language:message(l_sMessage,21)
      call use:type(l_nX,l_nY,l_sMessage)
      // read the new trajectory
      call use:read(l_nX+len(l_sMessage),l_nY,l_sName,10,false)
      if !use:bUseEscape
        // look if the items exist
        call new(l_sName,l_nResult)
        if l_nResult==-1
          call language:message(l_sMessage,-2)
          popUpMsg(l_sMessage)
        endIf
      endIf
    break
  endSwitch
  if l_nKey!=255
    x_sItem=l_sName
  else
    x_sItem=""
  endIf
end

--- onProgEnd.pgx ---
public program onProgEnd(string& x_sItem[])
begin
end

--- onRun.pgx ---
public program onRun(string& x_sItem[])
  local string l_sEmpty
  local num l_nResult
begin
  // execute check if need to reload
  call loadCycle(x_sItem,l_nResult)
  // execute
  call makeTraj(x_sItem)
end

--- onSave.pgx ---
public program onSave(string& x_sItem[])
  local num i
  local num l_nSize
begin
  //if bToSave
  // update
  if isDefined(pt:tTraj[pEditPoint.sID])
    pt:tTraj[pEditPoint.sID]=pEditPoint
    call pt:link_all(pEditPoint.sID)
  endIf
  // saveIt
  pt:libSave()
  bToSave=false
  //$fileClose(nFile)
  // endIf
end

--- onStart.pgx ---
public program onStart(string& x_sItem[])
  local num i
  local string l_sType
begin

end

--- onStop.pgx ---
public program onStop(string& x_sItem[])
begin
  // stop it
  if x_sItem=="kill"
    pt:libLoad("Disk://kernel/template/session/saveTraj/TRAJ")
  endIf
end

--- setFrameId.pgx ---
public program setFrameId(num x_nIndex)
  local num i
begin
  //
  // save the FrameId
  //
  pEditPoint.nIndexFrame=x_nIndex
  // link to the father frame
  pEditPoint.fFrame.trsf=saveData:fFrameItem[x_nIndex].fFrame.trsf
  for i=0 to size(pEditPoint.tData)-1
    link(pEditPoint.tData[i].pPoint,pEditPoint.fFrame)
  endFor
end

--- setTrajItem.pgx ---
public program setTrajItem(TrajectoryItem& x_tTraj[], num x_nIndex)
begin
  //
  // set all the field
  //
  pEditPoint.tData[x_nIndex].tSuper=x_tTraj
  // active the save data
  bToSave=true
end
